(* Logix 5000 project; controller PRU vendor 1 type 14 code 107 rev 20.13; software revision 20.01; part 6 of 17 *)
(* tags used below, declared in another part *)
   AFI : BOOL;
   AlarmMaster : DINT;
   AlarmMasterDisable : BOOL;
   AlarmMasterResetTON : TIMER;
   AlarmResetPB : BOOL;
   ALL_SHUTDOWN_FAULTS_IOK : BOOL;
   DRYER : DUAL_SCREW;
   DRYER_CENTER_STARTUP_MODE : BOOL;
   DRYER_MODE_AUTO : BOOL;
   ENCODER_ERROR : REAL;
   ESR_CONTACT_1_ION : BOOL;
   ESR_CONTACT_2_ION : BOOL;
   ESTOP_PB_IOF : BOOL;   // E-STOP PUSHBUTTON IS PUSHED.
   FAULT : DINT[100];
   FAULT_TIMER : TIMER[10000];
   FS0101_ION : BOOL;   // LOW FLOW SWITCH - INLET AND DISCHARGE PURGE
   FS0102H_ION : BOOL;   // HIGH FLOW SWITCH - DISCHARGE END SHAFT SEAL
   FS0102L_ION : BOOL;   // LOW FLOW SWITCH - DISCHARGE END SHAFT SEAL
   FS0103H_ION : BOOL;   // HIGH FLOW SWITCH - CHAMBER END INLET SEALS
   FS0103L_ION : BOOL;   // LOW FLOW SWITCH - CHAMBER END INLET SEALS
   FS0201_ION : BOOL;   // LOW FLOW SWITCH - KG021 PURGE
   FS0202_ION : BOOL;   // LOW FLOW SWITCH - KG022 PURGE
   FS0203H_ION : BOOL;   // HIGH FLOW SWITCH - COOLING SHAFT SEALS
   FS0203L_ION : BOOL;   // LOW FLOW SWITCH - COOLING SHAFT SEALS
   FS0204_ION : BOOL;   // LOW FLOW SWITCH - COOLING SCREW COOLING WATER
   HMI_ALARM_RESET : BOOL;
   HMI_FINAL_SCREW_POSITION_ERROR : REAL;
   K0621_IS_LOCAL : BOOL;
   K0621_IS_REMOTE : BOOL;
   K0622_IS_LOCAL : BOOL;
   K0622_IS_REMOTE : BOOL;
   MAX_ENCODER_ERROR_MINUS_WARN : REAL;
   MAX_ENCODER_ERROR_PLUS_WARN : REAL;
   PS0101_ION : BOOL;   // PRESSURE SWITCH - CONTROL PANEL Y/Z N2 PURGE
   PS0102_ION : BOOL;   // PRESSURE SWITCH - MAIN N2 SUPPLY
   SCREWS_ENABLE_GON : BOOL;   // Dryer screw faults are ok.
   SV0101 : BOOL;
   SV0102 : BOOL;
   SV0201 : BOOL;
   SV0202 : BOOL;
   SV0203 : BOOL;
   TE0101 : REAL;
   TE0102 : REAL;
   TE0103 : REAL;
   TE0104 : REAL;
   TE0105 : REAL;
   TE0106 : REAL;
   TE0107 : REAL;
   TE0108 : REAL;
   TE0109 : REAL;
   TE0110 : REAL;
   TE0111 : REAL;
   TE0112 : REAL;
   TE0113 : REAL;
   TE0114 : REAL;
   TE0115 : REAL;
   TE0116 : REAL;
   TE0117 : REAL;
   TE0118 : REAL;
   TE0119 : REAL;
   TE0120 : REAL;
   TE0121 : REAL;
   TE0122 : REAL;
   TE0123 : REAL;
   TE0124 : REAL;
   TE0125 : REAL;
   TE0126 : REAL;
   TE0127 : REAL;
   TE0128 : REAL;
   TE0129 : REAL;
   TE0130 : REAL;
   TE0201 : REAL;
   TE0202 : REAL;
   THRESHOLD : REAL[9000];
   VFD_1_Current_Real : REAL;
   VFD_2_Current_Real : REAL;
   VFD_3_Current_Real : REAL;
   VFDS_BON : BOOL;   // DRYER VFDs HAVE BEEN COMMANDED ON FOR 1 SECOND.
   WARNA_IOK : BOOL;
   WARND_IOK : BOOL;
   WARNE_IOK : BOOL;
   WIPE_ACTUAL : REAL;
(* MainProgram, continued *)

ROUTINE A4_Alarms_General   (* ladder *)
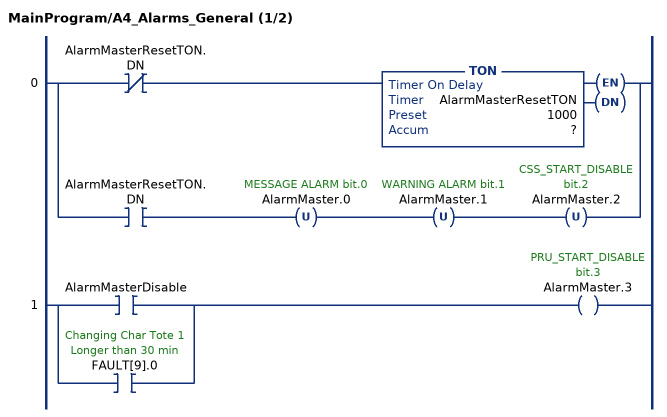
   0: [XIO(AlarmMasterResetTON.DN) TON(AlarmMasterResetTON,?,?) ,XIC(AlarmMasterResetTON.DN) OTU(AlarmMaster.0) OTU(AlarmMaster.1) OTU(AlarmMaster.2) ];
   1: [XIC(AlarmMasterDisable) ,XIC(FAULT[9].0) ]OTE(AlarmMaster.3);
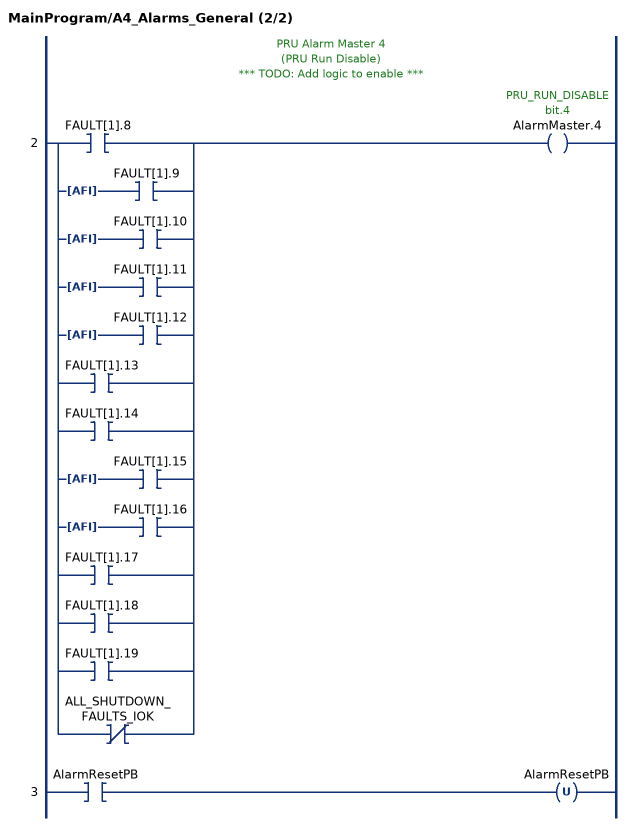
   // PRU Alarm Master 4
   // (PRU Run Disable)
   // *** TODO: Add logic to enable ***
   2: [XIC(FAULT[1].8) ,AFI() XIC(FAULT[1].9) ,AFI() XIC(FAULT[1].10) ,AFI() XIC(FAULT[1].11) ,AFI() XIC(FAULT[1].12) ,XIC(FAULT[1].13) ,XIC(FAULT[1].14) ,AFI() XIC(FAULT[1].15) ,AFI() XIC(FAULT[1].16) ,XIC(FAULT[1].17) ,XIC(FAULT[1].18) ,XIC(FAULT[1].19) ,XIO(ALL_SHUTDOWN_FAULTS_IOK) ]OTE(AlarmMaster.4);
   3: XIC(AlarmResetPB)OTU(AlarmResetPB);
END_ROUTINE

ROUTINE B00_WARN_A_100   (* ladder *)
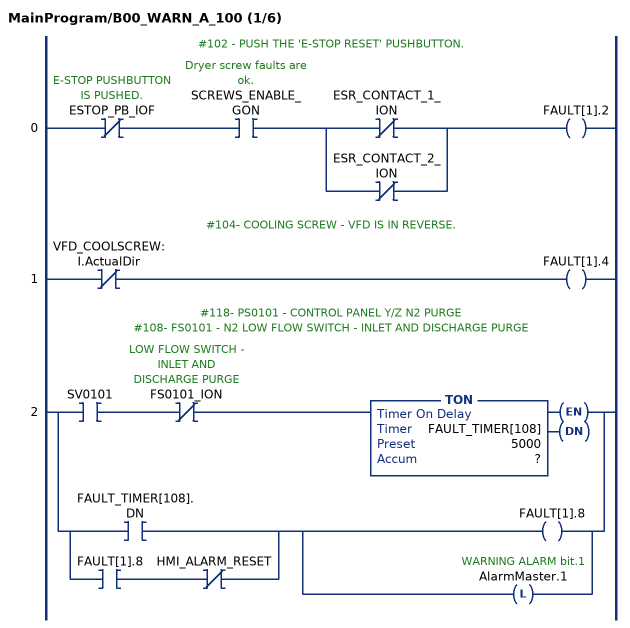
   // #102 - PUSH THE 'E-STOP RESET' PUSHBUTTON.
   0: XIO(ESTOP_PB_IOF)XIC(SCREWS_ENABLE_GON)[XIO(ESR_CONTACT_1_ION) ,XIO(ESR_CONTACT_2_ION) ]OTE(FAULT[1].2);
   // #104- COOLING SCREW - VFD IS IN REVERSE.
   1: XIO(VFD_COOLSCREW:I.ActualDir)OTE(FAULT[1].4);
   // #118- PS0101 - CONTROL PANEL Y/Z N2 PURGE
   // #108- FS0101 - N2 LOW FLOW SWITCH - INLET AND DISCHARGE PURGE
   2: [XIC(SV0101) XIO(FS0101_ION) TON(FAULT_TIMER[108],?,?) ,[XIC(FAULT_TIMER[108].DN) ,XIC(FAULT[1].8) XIO(HMI_ALARM_RESET) ] [OTE(FAULT[1].8) ,OTL(AlarmMaster.1) ] ];
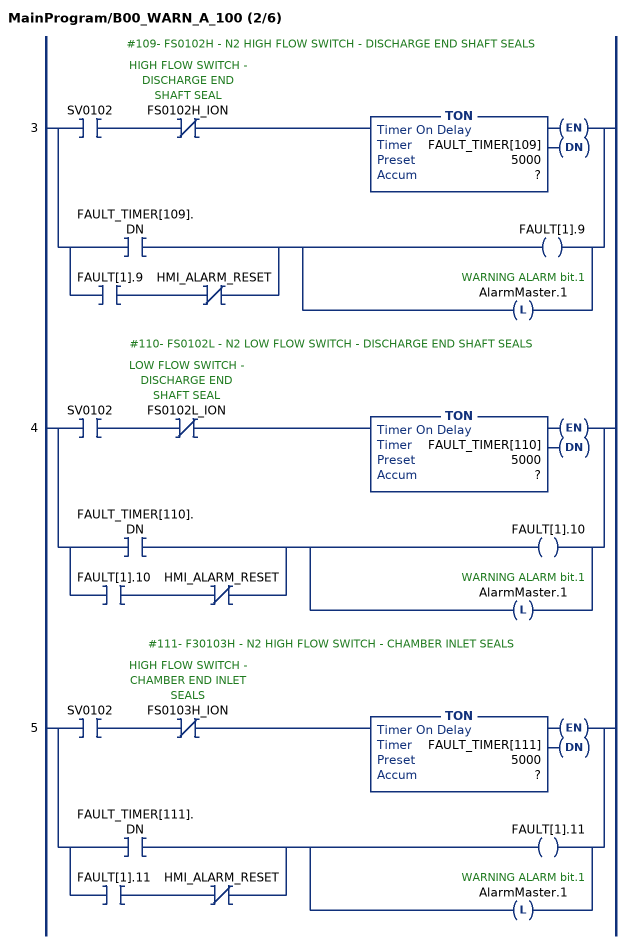
   // #109- FS0102H - N2 HIGH FLOW SWITCH - DISCHARGE END SHAFT SEALS
   3: [XIC(SV0102) XIO(FS0102H_ION) TON(FAULT_TIMER[109],?,?) ,[XIC(FAULT_TIMER[109].DN) ,XIC(FAULT[1].9) XIO(HMI_ALARM_RESET) ] [OTE(FAULT[1].9) ,OTL(AlarmMaster.1) ] ];
   // #110- FS0102L - N2 LOW FLOW SWITCH - DISCHARGE END SHAFT SEALS
   4: [XIC(SV0102) XIO(FS0102L_ION) TON(FAULT_TIMER[110],?,?) ,[XIC(FAULT_TIMER[110].DN) ,XIC(FAULT[1].10) XIO(HMI_ALARM_RESET) ] [OTE(FAULT[1].10) ,OTL(AlarmMaster.1) ] ];
   // #111- F30103H - N2 HIGH FLOW SWITCH - CHAMBER INLET SEALS
   5: [XIC(SV0102) XIO(FS0103H_ION) TON(FAULT_TIMER[111],?,?) ,[XIC(FAULT_TIMER[111].DN) ,XIC(FAULT[1].11) XIO(HMI_ALARM_RESET) ] [OTE(FAULT[1].11) ,OTL(AlarmMaster.1) ] ];
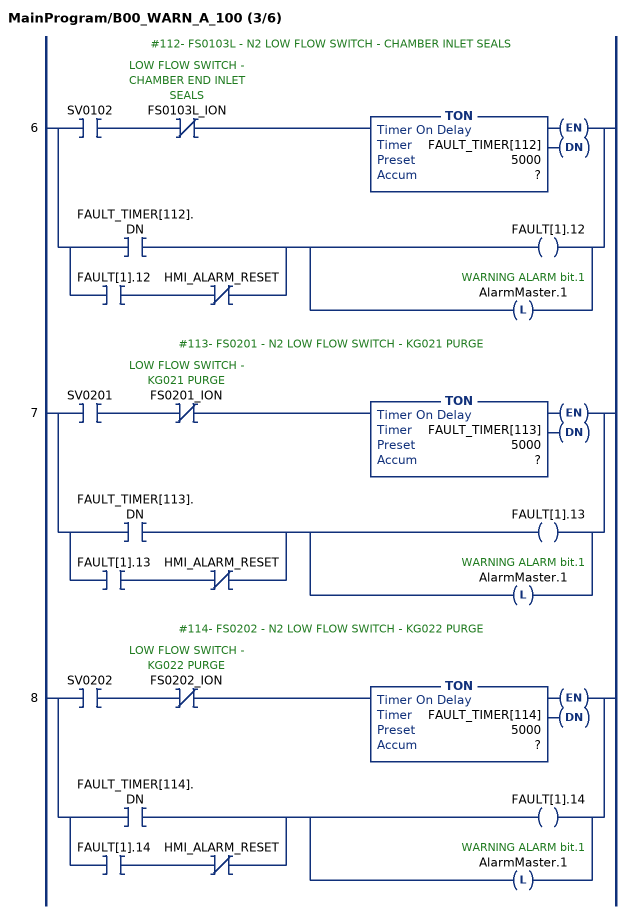
   // #112- FS0103L - N2 LOW FLOW SWITCH - CHAMBER INLET SEALS
   6: [XIC(SV0102) XIO(FS0103L_ION) TON(FAULT_TIMER[112],?,?) ,[XIC(FAULT_TIMER[112].DN) ,XIC(FAULT[1].12) XIO(HMI_ALARM_RESET) ] [OTE(FAULT[1].12) ,OTL(AlarmMaster.1) ] ];
   // #113- FS0201 - N2 LOW FLOW SWITCH - KG021 PURGE
   7: [XIC(SV0201) XIO(FS0201_ION) TON(FAULT_TIMER[113],?,?) ,[XIC(FAULT_TIMER[113].DN) ,XIC(FAULT[1].13) XIO(HMI_ALARM_RESET) ] [OTE(FAULT[1].13) ,OTL(AlarmMaster.1) ] ];
   // #114- FS0202 - N2 LOW FLOW SWITCH - KG022 PURGE
   8: [XIC(SV0202) XIO(FS0202_ION) TON(FAULT_TIMER[114],?,?) ,[XIC(FAULT_TIMER[114].DN) ,XIC(FAULT[1].14) XIO(HMI_ALARM_RESET) ] [OTE(FAULT[1].14) ,OTL(AlarmMaster.1) ] ];
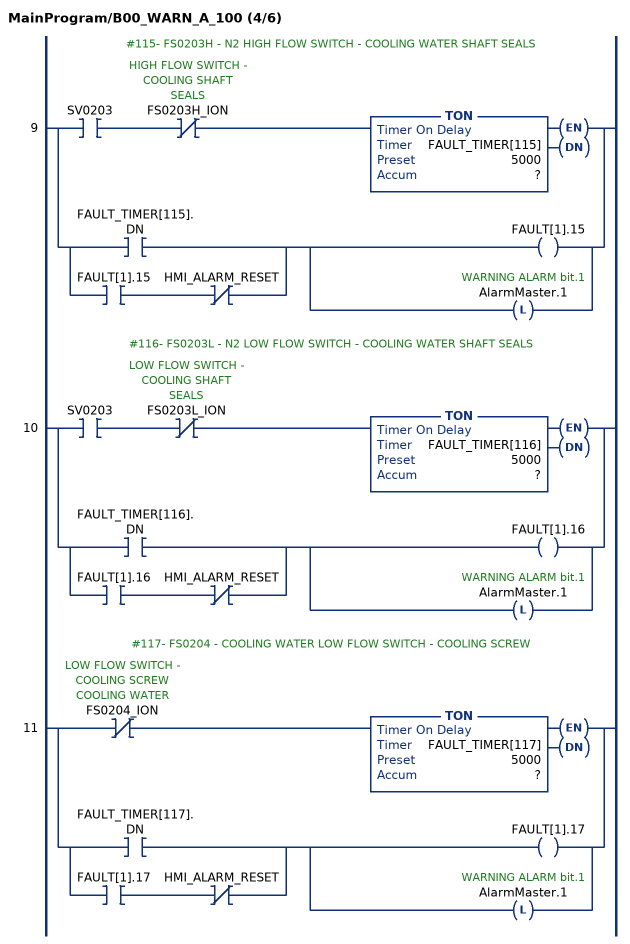
   // #115- FS0203H - N2 HIGH FLOW SWITCH - COOLING WATER SHAFT SEALS
   9: [XIC(SV0203) XIO(FS0203H_ION) TON(FAULT_TIMER[115],?,?) ,[XIC(FAULT_TIMER[115].DN) ,XIC(FAULT[1].15) XIO(HMI_ALARM_RESET) ] [OTE(FAULT[1].15) ,OTL(AlarmMaster.1) ] ];
   // #116- FS0203L - N2 LOW FLOW SWITCH - COOLING WATER SHAFT SEALS
   10: [XIC(SV0203) XIO(FS0203L_ION) TON(FAULT_TIMER[116],?,?) ,[XIC(FAULT_TIMER[116].DN) ,XIC(FAULT[1].16) XIO(HMI_ALARM_RESET) ] [OTE(FAULT[1].16) ,OTL(AlarmMaster.1) ] ];
   // #117- FS0204 - COOLING WATER LOW FLOW SWITCH - COOLING SCREW
   11: [XIO(FS0204_ION) TON(FAULT_TIMER[117],?,?) ,[XIC(FAULT_TIMER[117].DN) ,XIC(FAULT[1].17) XIO(HMI_ALARM_RESET) ] [OTE(FAULT[1].17) ,OTL(AlarmMaster.1) ] ];
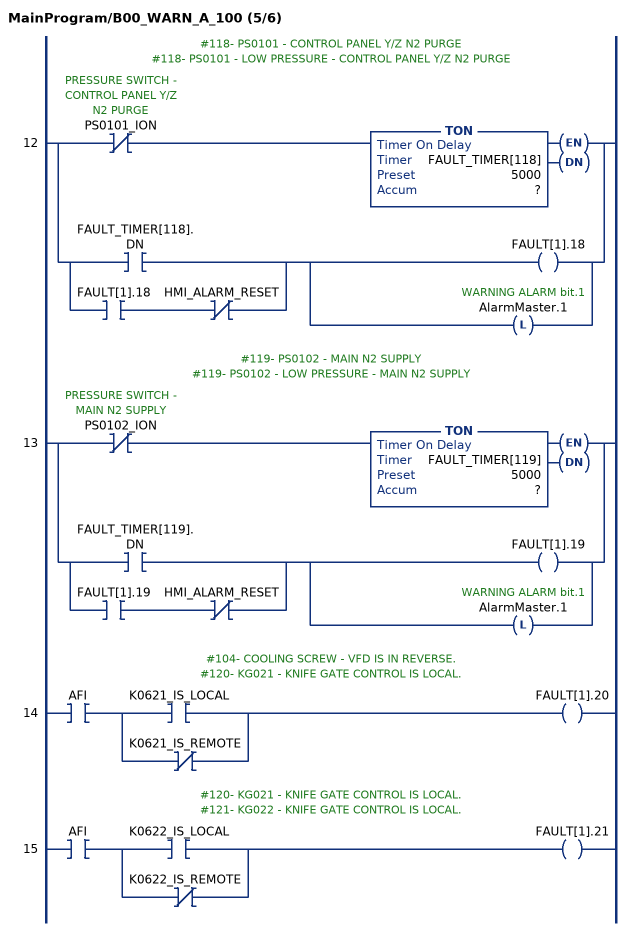
   // #118- PS0101 - CONTROL PANEL Y/Z N2 PURGE
   // #118- PS0101 - LOW PRESSURE - CONTROL PANEL Y/Z N2 PURGE
   12: [XIO(PS0101_ION) TON(FAULT_TIMER[118],?,?) ,[XIC(FAULT_TIMER[118].DN) ,XIC(FAULT[1].18) XIO(HMI_ALARM_RESET) ] [OTE(FAULT[1].18) ,OTL(AlarmMaster.1) ] ];
   // #119- PS0102 - MAIN N2 SUPPLY
   // #119- PS0102 - LOW PRESSURE - MAIN N2 SUPPLY
   13: [XIO(PS0102_ION) TON(FAULT_TIMER[119],?,?) ,[XIC(FAULT_TIMER[119].DN) ,XIC(FAULT[1].19) XIO(HMI_ALARM_RESET) ] [OTE(FAULT[1].19) ,OTL(AlarmMaster.1) ] ];
   // #104- COOLING SCREW - VFD IS IN REVERSE.
   // #120- KG021 - KNIFE GATE CONTROL IS LOCAL.
   14: XIC(AFI)[XIC(K0621_IS_LOCAL) ,XIO(K0621_IS_REMOTE) ]OTE(FAULT[1].20);
   // #120- KG021 - KNIFE GATE CONTROL IS LOCAL.
   // #121- KG022 - KNIFE GATE CONTROL IS LOCAL.
   15: XIC(AFI)[XIC(K0622_IS_LOCAL) ,XIO(K0622_IS_REMOTE) ]OTE(FAULT[1].21);
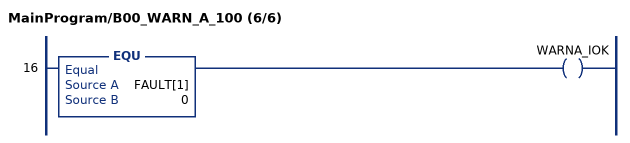
   16: EQU(FAULT[1],0)OTE(WARNA_IOK);
END_ROUTINE

ROUTINE B00_WARN_D_400_CURRENT   (* ladder *)
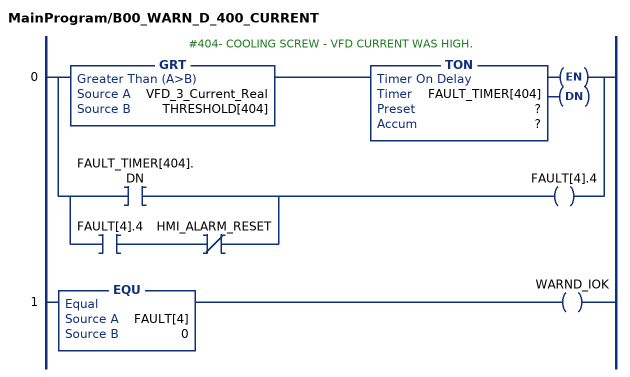
   // #404- COOLING SCREW - VFD CURRENT WAS HIGH.
   0: [GRT(VFD_3_Current_Real,THRESHOLD[404]) TON(FAULT_TIMER[404],?,?) ,[XIC(FAULT_TIMER[404].DN) ,XIC(FAULT[4].4) XIO(HMI_ALARM_RESET) ] OTE(FAULT[4].4) ];
   1: EQU(FAULT[4],0)OTE(WARND_IOK);
END_ROUTINE

ROUTINE B00_WARN_E_500_DRYER   (* ladder *)
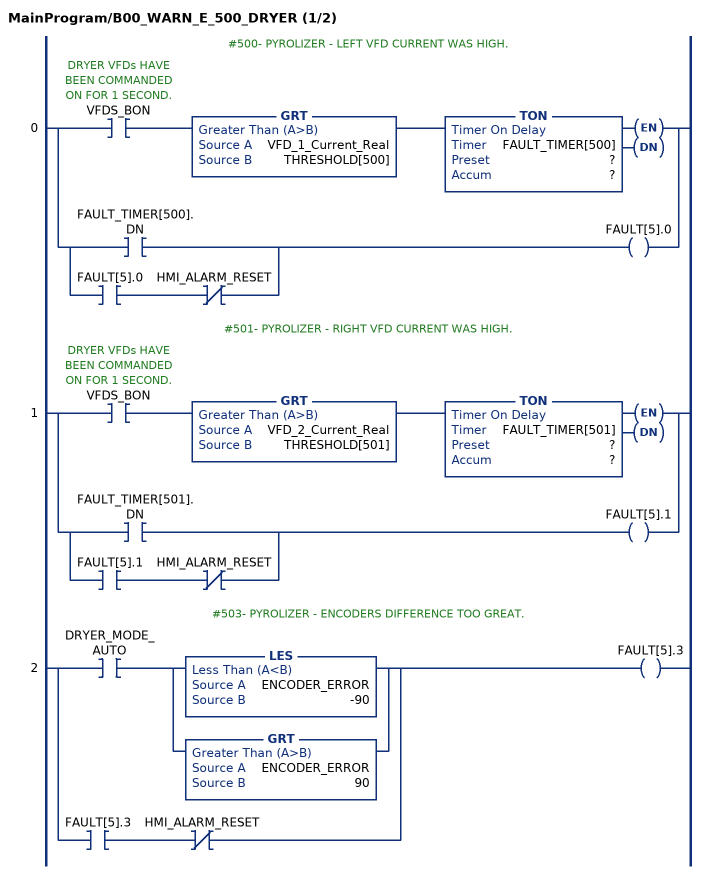
   // #500- PYROLIZER - LEFT VFD CURRENT WAS HIGH.
   0: [XIC(VFDS_BON) GRT(VFD_1_Current_Real,THRESHOLD[500]) TON(FAULT_TIMER[500],?,?) ,[XIC(FAULT_TIMER[500].DN) ,XIC(FAULT[5].0) XIO(HMI_ALARM_RESET) ] OTE(FAULT[5].0) ];
   // #501- PYROLIZER - RIGHT VFD CURRENT WAS HIGH.
   1: [XIC(VFDS_BON) GRT(VFD_2_Current_Real,THRESHOLD[501]) TON(FAULT_TIMER[501],?,?) ,[XIC(FAULT_TIMER[501].DN) ,XIC(FAULT[5].1) XIO(HMI_ALARM_RESET) ] OTE(FAULT[5].1) ];
   // #503- PYROLIZER - ENCODERS DIFFERENCE TOO GREAT.
   2: [XIC(DRYER_MODE_AUTO) [LES(ENCODER_ERROR,-90) ,GRT(ENCODER_ERROR,90) ] ,XIC(FAULT[5].3) XIO(HMI_ALARM_RESET) ]OTE(FAULT[5].3);
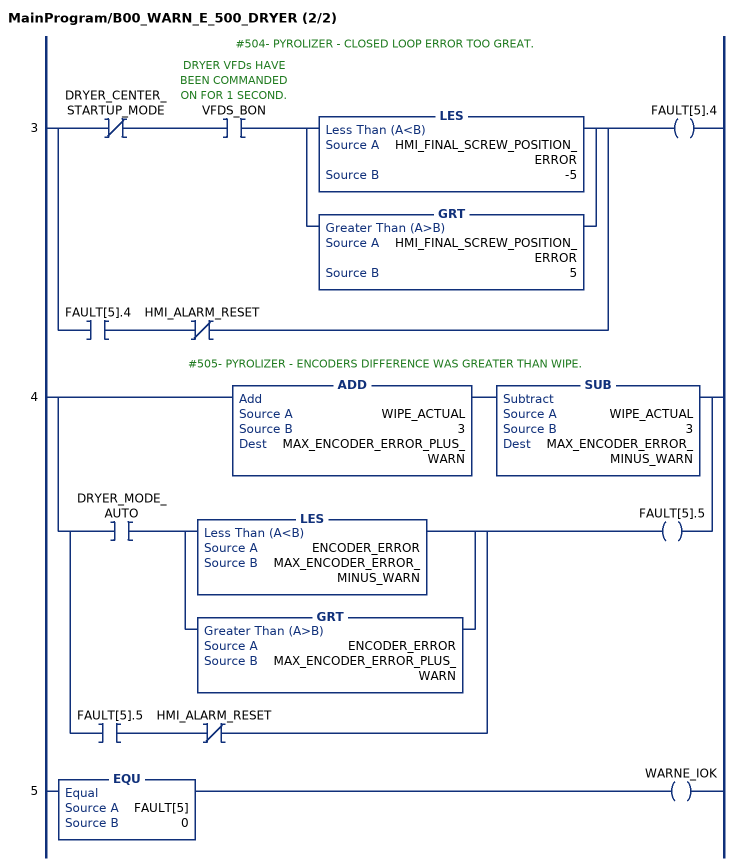
   // #504- PYROLIZER - CLOSED LOOP ERROR TOO GREAT.
   3: [XIO(DRYER_CENTER_STARTUP_MODE) XIC(VFDS_BON) [LES(HMI_FINAL_SCREW_POSITION_ERROR,-5) ,GRT(HMI_FINAL_SCREW_POSITION_ERROR,5) ] ,XIC(FAULT[5].4) XIO(HMI_ALARM_RESET) ]OTE(FAULT[5].4);
   // #505- PYROLIZER - ENCODERS DIFFERENCE WAS GREATER THAN WIPE.
   4: [ADD(WIPE_ACTUAL,3,MAX_ENCODER_ERROR_PLUS_WARN) SUB(WIPE_ACTUAL,3,MAX_ENCODER_ERROR_MINUS_WARN) ,[XIC(DRYER_MODE_AUTO) [LES(ENCODER_ERROR,MAX_ENCODER_ERROR_MINUS_WARN) ,GRT(ENCODER_ERROR,MAX_ENCODER_ERROR_PLUS_WARN) ] ,XIC(FAULT[5].5) XIO(HMI_ALARM_RESET) ] OTE(FAULT[5].5) ];
   5: EQU(FAULT[5],0)OTE(WARNE_IOK);
END_ROUTINE

ROUTINE B00_WARN_F_600_HI_TEMP   (* ladder *)
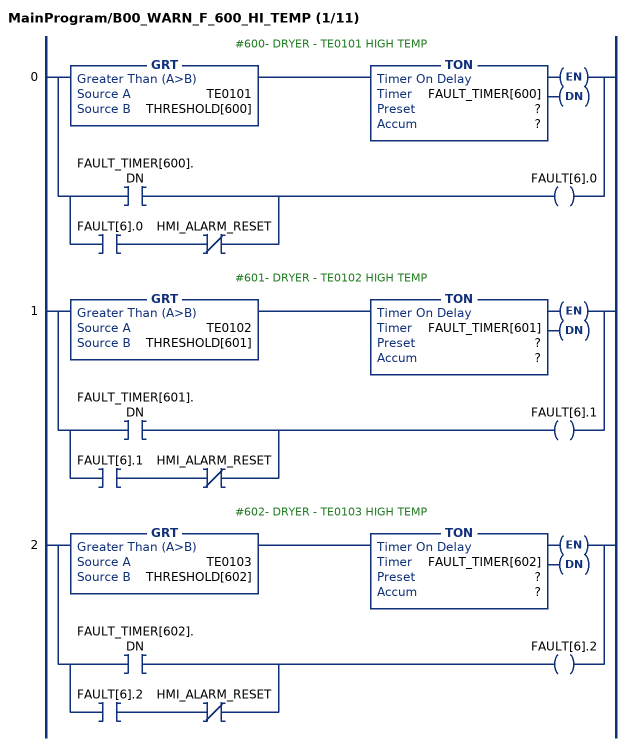
   // #600- DRYER - TE0101 HIGH TEMP
   0: [GRT(TE0101,THRESHOLD[600]) TON(FAULT_TIMER[600],?,?) ,[XIC(FAULT_TIMER[600].DN) ,XIC(FAULT[6].0) XIO(HMI_ALARM_RESET) ] OTE(FAULT[6].0) ];
   // #601- DRYER - TE0102 HIGH TEMP
   1: [GRT(TE0102,THRESHOLD[601]) TON(FAULT_TIMER[601],?,?) ,[XIC(FAULT_TIMER[601].DN) ,XIC(FAULT[6].1) XIO(HMI_ALARM_RESET) ] OTE(FAULT[6].1) ];
   // #602- DRYER - TE0103 HIGH TEMP
   2: [GRT(TE0103,THRESHOLD[602]) TON(FAULT_TIMER[602],?,?) ,[XIC(FAULT_TIMER[602].DN) ,XIC(FAULT[6].2) XIO(HMI_ALARM_RESET) ] OTE(FAULT[6].2) ];
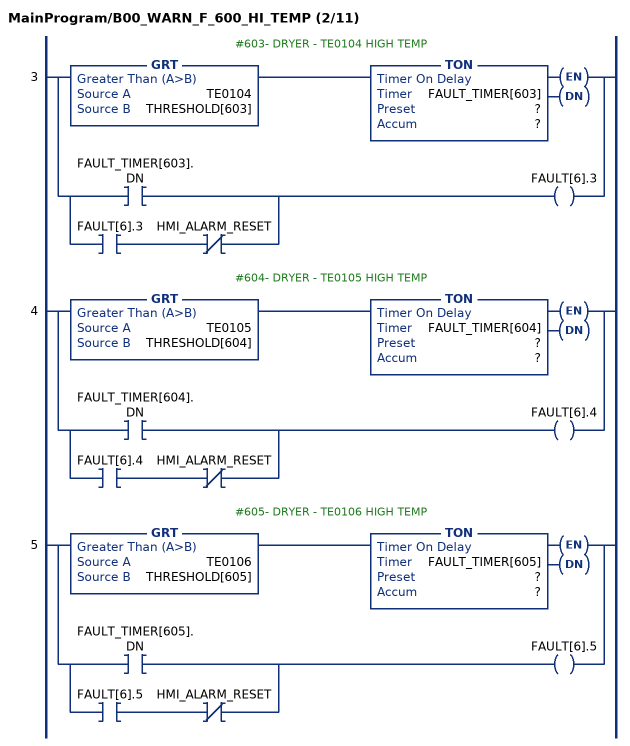
   // #603- DRYER - TE0104 HIGH TEMP
   3: [GRT(TE0104,THRESHOLD[603]) TON(FAULT_TIMER[603],?,?) ,[XIC(FAULT_TIMER[603].DN) ,XIC(FAULT[6].3) XIO(HMI_ALARM_RESET) ] OTE(FAULT[6].3) ];
   // #604- DRYER - TE0105 HIGH TEMP
   4: [GRT(TE0105,THRESHOLD[604]) TON(FAULT_TIMER[604],?,?) ,[XIC(FAULT_TIMER[604].DN) ,XIC(FAULT[6].4) XIO(HMI_ALARM_RESET) ] OTE(FAULT[6].4) ];
   // #605- DRYER - TE0106 HIGH TEMP
   5: [GRT(TE0106,THRESHOLD[605]) TON(FAULT_TIMER[605],?,?) ,[XIC(FAULT_TIMER[605].DN) ,XIC(FAULT[6].5) XIO(HMI_ALARM_RESET) ] OTE(FAULT[6].5) ];
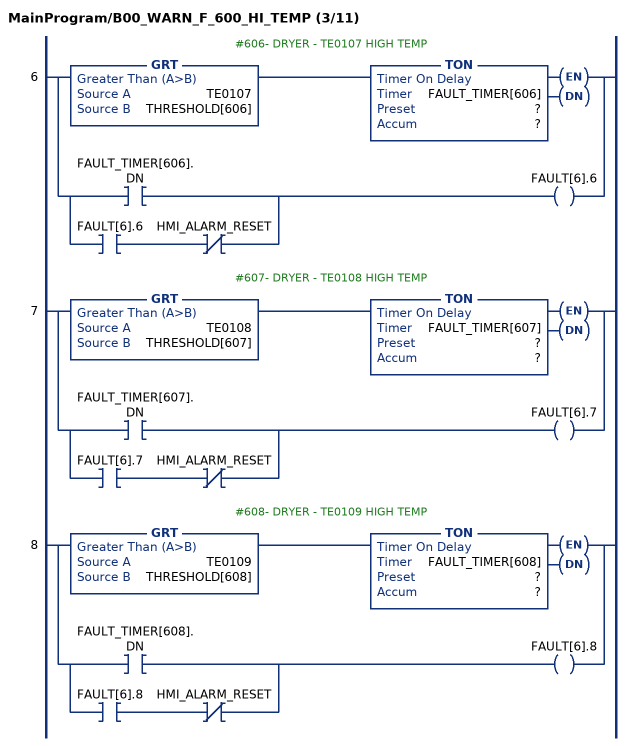
   // #606- DRYER - TE0107 HIGH TEMP
   6: [GRT(TE0107,THRESHOLD[606]) TON(FAULT_TIMER[606],?,?) ,[XIC(FAULT_TIMER[606].DN) ,XIC(FAULT[6].6) XIO(HMI_ALARM_RESET) ] OTE(FAULT[6].6) ];
   // #607- DRYER - TE0108 HIGH TEMP
   7: [GRT(TE0108,THRESHOLD[607]) TON(FAULT_TIMER[607],?,?) ,[XIC(FAULT_TIMER[607].DN) ,XIC(FAULT[6].7) XIO(HMI_ALARM_RESET) ] OTE(FAULT[6].7) ];
   // #608- DRYER - TE0109 HIGH TEMP
   8: [GRT(TE0109,THRESHOLD[608]) TON(FAULT_TIMER[608],?,?) ,[XIC(FAULT_TIMER[608].DN) ,XIC(FAULT[6].8) XIO(HMI_ALARM_RESET) ] OTE(FAULT[6].8) ];
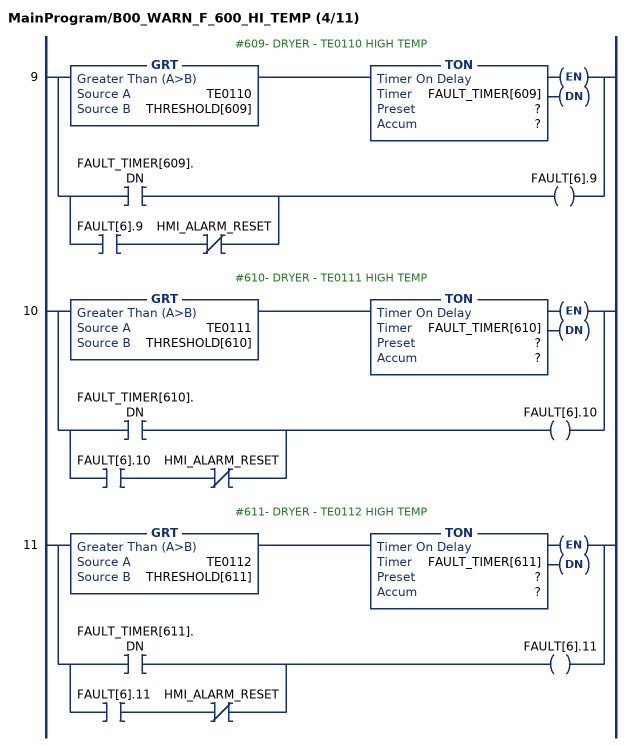
   // #609- DRYER - TE0110 HIGH TEMP
   9: [GRT(TE0110,THRESHOLD[609]) TON(FAULT_TIMER[609],?,?) ,[XIC(FAULT_TIMER[609].DN) ,XIC(FAULT[6].9) XIO(HMI_ALARM_RESET) ] OTE(FAULT[6].9) ];
   // #610- DRYER - TE0111 HIGH TEMP
   10: [GRT(TE0111,THRESHOLD[610]) TON(FAULT_TIMER[610],?,?) ,[XIC(FAULT_TIMER[610].DN) ,XIC(FAULT[6].10) XIO(HMI_ALARM_RESET) ] OTE(FAULT[6].10) ];
   // #611- DRYER - TE0112 HIGH TEMP
   11: [GRT(TE0112,THRESHOLD[611]) TON(FAULT_TIMER[611],?,?) ,[XIC(FAULT_TIMER[611].DN) ,XIC(FAULT[6].11) XIO(HMI_ALARM_RESET) ] OTE(FAULT[6].11) ];
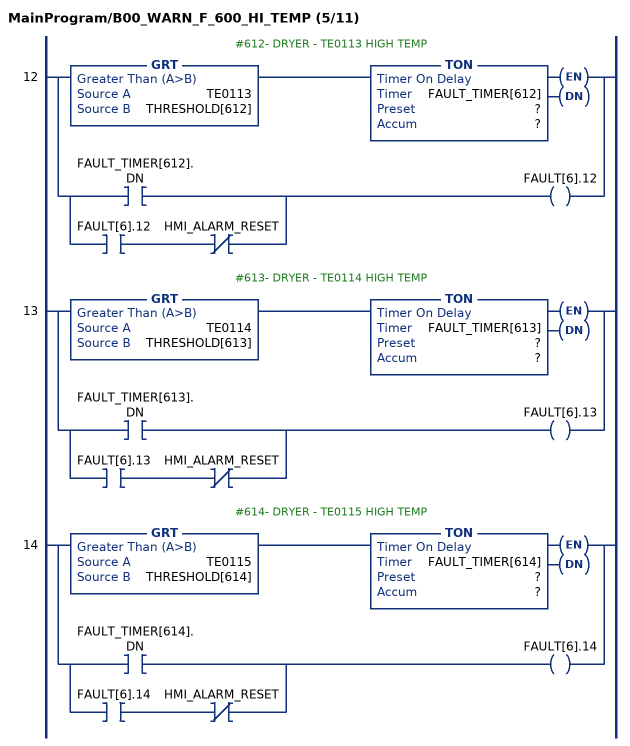
   // #612- DRYER - TE0113 HIGH TEMP
   12: [GRT(TE0113,THRESHOLD[612]) TON(FAULT_TIMER[612],?,?) ,[XIC(FAULT_TIMER[612].DN) ,XIC(FAULT[6].12) XIO(HMI_ALARM_RESET) ] OTE(FAULT[6].12) ];
   // #613- DRYER - TE0114 HIGH TEMP
   13: [GRT(TE0114,THRESHOLD[613]) TON(FAULT_TIMER[613],?,?) ,[XIC(FAULT_TIMER[613].DN) ,XIC(FAULT[6].13) XIO(HMI_ALARM_RESET) ] OTE(FAULT[6].13) ];
   // #614- DRYER - TE0115 HIGH TEMP
   14: [GRT(TE0115,THRESHOLD[614]) TON(FAULT_TIMER[614],?,?) ,[XIC(FAULT_TIMER[614].DN) ,XIC(FAULT[6].14) XIO(HMI_ALARM_RESET) ] OTE(FAULT[6].14) ];
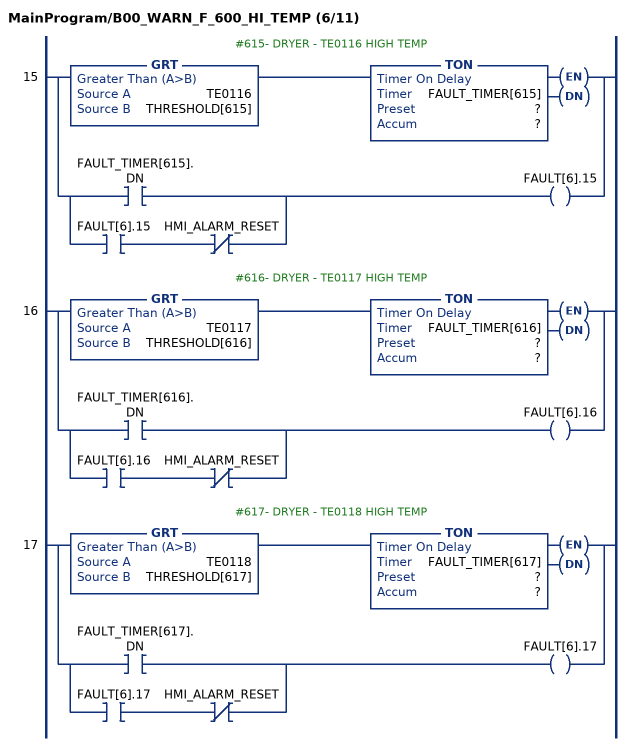
   // #615- DRYER - TE0116 HIGH TEMP
   15: [GRT(TE0116,THRESHOLD[615]) TON(FAULT_TIMER[615],?,?) ,[XIC(FAULT_TIMER[615].DN) ,XIC(FAULT[6].15) XIO(HMI_ALARM_RESET) ] OTE(FAULT[6].15) ];
   // #616- DRYER - TE0117 HIGH TEMP
   16: [GRT(TE0117,THRESHOLD[616]) TON(FAULT_TIMER[616],?,?) ,[XIC(FAULT_TIMER[616].DN) ,XIC(FAULT[6].16) XIO(HMI_ALARM_RESET) ] OTE(FAULT[6].16) ];
   // #617- DRYER - TE0118 HIGH TEMP
   17: [GRT(TE0118,THRESHOLD[617]) TON(FAULT_TIMER[617],?,?) ,[XIC(FAULT_TIMER[617].DN) ,XIC(FAULT[6].17) XIO(HMI_ALARM_RESET) ] OTE(FAULT[6].17) ];
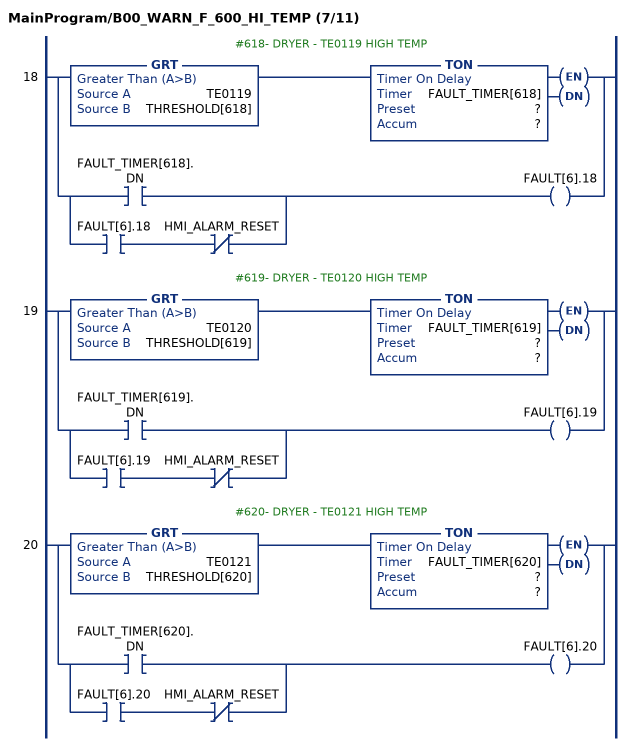
   // #618- DRYER - TE0119 HIGH TEMP
   18: [GRT(TE0119,THRESHOLD[618]) TON(FAULT_TIMER[618],?,?) ,[XIC(FAULT_TIMER[618].DN) ,XIC(FAULT[6].18) XIO(HMI_ALARM_RESET) ] OTE(FAULT[6].18) ];
   // #619- DRYER - TE0120 HIGH TEMP
   19: [GRT(TE0120,THRESHOLD[619]) TON(FAULT_TIMER[619],?,?) ,[XIC(FAULT_TIMER[619].DN) ,XIC(FAULT[6].19) XIO(HMI_ALARM_RESET) ] OTE(FAULT[6].19) ];
   // #620- DRYER - TE0121 HIGH TEMP
   20: [GRT(TE0121,THRESHOLD[620]) TON(FAULT_TIMER[620],?,?) ,[XIC(FAULT_TIMER[620].DN) ,XIC(FAULT[6].20) XIO(HMI_ALARM_RESET) ] OTE(FAULT[6].20) ];
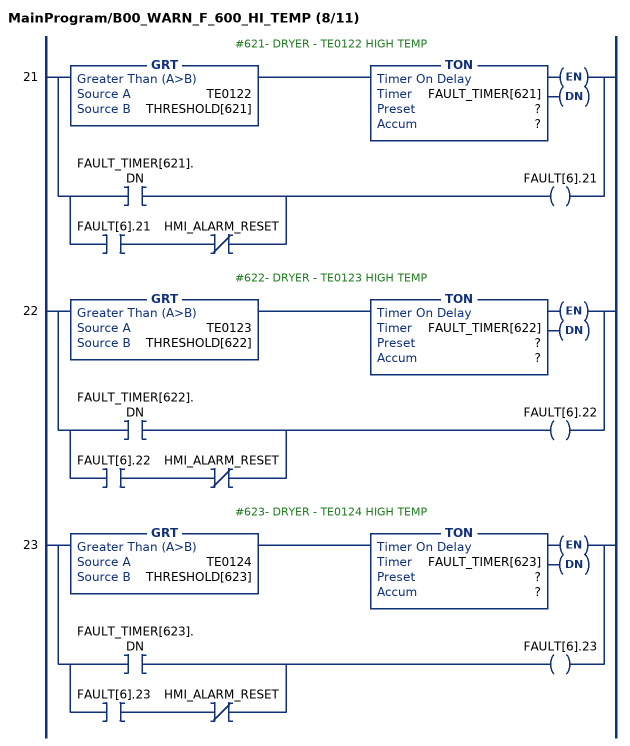
   // #621- DRYER - TE0122 HIGH TEMP
   21: [GRT(TE0122,THRESHOLD[621]) TON(FAULT_TIMER[621],?,?) ,[XIC(FAULT_TIMER[621].DN) ,XIC(FAULT[6].21) XIO(HMI_ALARM_RESET) ] OTE(FAULT[6].21) ];
   // #622- DRYER - TE0123 HIGH TEMP
   22: [GRT(TE0123,THRESHOLD[622]) TON(FAULT_TIMER[622],?,?) ,[XIC(FAULT_TIMER[622].DN) ,XIC(FAULT[6].22) XIO(HMI_ALARM_RESET) ] OTE(FAULT[6].22) ];
   // #623- DRYER - TE0124 HIGH TEMP
   23: [GRT(TE0124,THRESHOLD[623]) TON(FAULT_TIMER[623],?,?) ,[XIC(FAULT_TIMER[623].DN) ,XIC(FAULT[6].23) XIO(HMI_ALARM_RESET) ] OTE(FAULT[6].23) ];
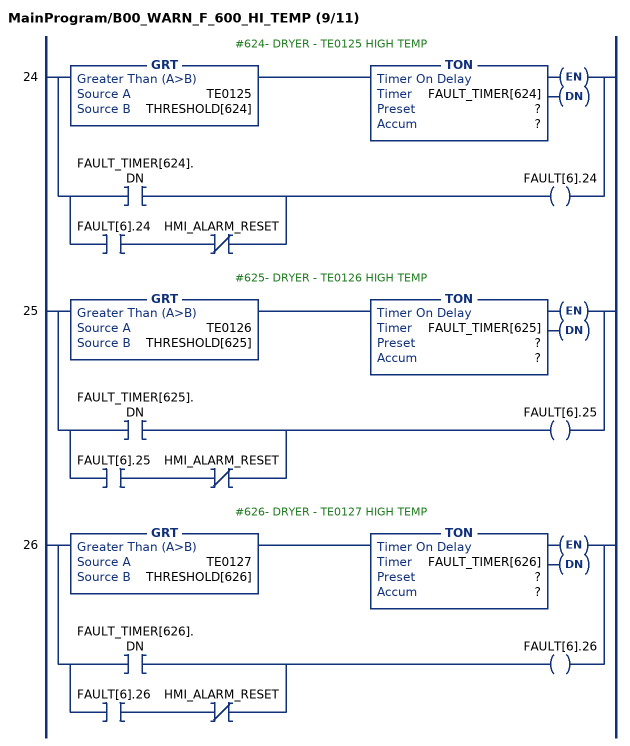
   // #624- DRYER - TE0125 HIGH TEMP
   24: [GRT(TE0125,THRESHOLD[624]) TON(FAULT_TIMER[624],?,?) ,[XIC(FAULT_TIMER[624].DN) ,XIC(FAULT[6].24) XIO(HMI_ALARM_RESET) ] OTE(FAULT[6].24) ];
   // #625- DRYER - TE0126 HIGH TEMP
   25: [GRT(TE0126,THRESHOLD[625]) TON(FAULT_TIMER[625],?,?) ,[XIC(FAULT_TIMER[625].DN) ,XIC(FAULT[6].25) XIO(HMI_ALARM_RESET) ] OTE(FAULT[6].25) ];
   // #626- DRYER - TE0127 HIGH TEMP
   26: [GRT(TE0127,THRESHOLD[626]) TON(FAULT_TIMER[626],?,?) ,[XIC(FAULT_TIMER[626].DN) ,XIC(FAULT[6].26) XIO(HMI_ALARM_RESET) ] OTE(FAULT[6].26) ];
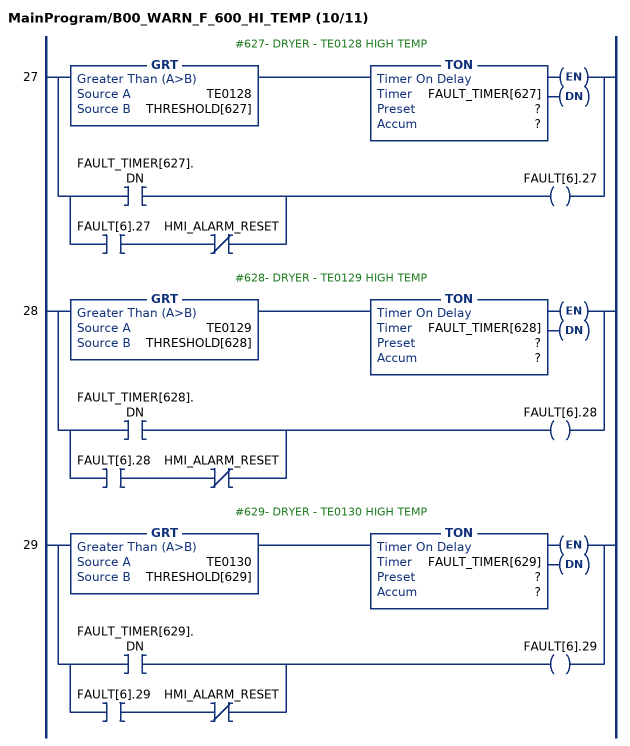
   // #627- DRYER - TE0128 HIGH TEMP
   27: [GRT(TE0128,THRESHOLD[627]) TON(FAULT_TIMER[627],?,?) ,[XIC(FAULT_TIMER[627].DN) ,XIC(FAULT[6].27) XIO(HMI_ALARM_RESET) ] OTE(FAULT[6].27) ];
   // #628- DRYER - TE0129 HIGH TEMP
   28: [GRT(TE0129,THRESHOLD[628]) TON(FAULT_TIMER[628],?,?) ,[XIC(FAULT_TIMER[628].DN) ,XIC(FAULT[6].28) XIO(HMI_ALARM_RESET) ] OTE(FAULT[6].28) ];
   // #629- DRYER - TE0130 HIGH TEMP
   29: [GRT(TE0130,THRESHOLD[629]) TON(FAULT_TIMER[629],?,?) ,[XIC(FAULT_TIMER[629].DN) ,XIC(FAULT[6].29) XIO(HMI_ALARM_RESET) ] OTE(FAULT[6].29) ];
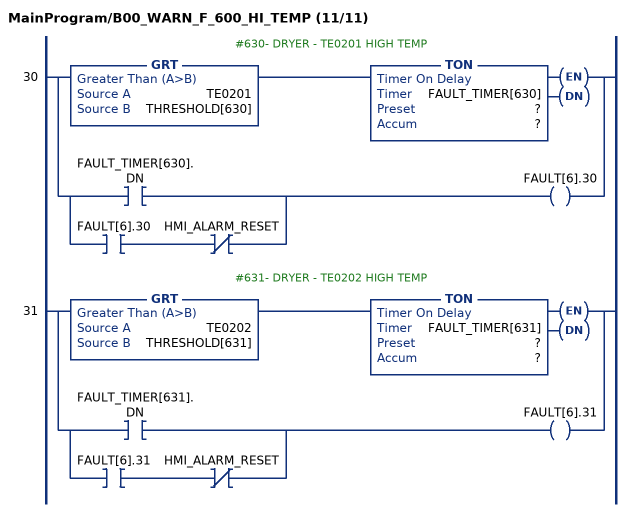
   // #630- DRYER - TE0201 HIGH TEMP
   30: [GRT(TE0201,THRESHOLD[630]) TON(FAULT_TIMER[630],?,?) ,[XIC(FAULT_TIMER[630].DN) ,XIC(FAULT[6].30) XIO(HMI_ALARM_RESET) ] OTE(FAULT[6].30) ];
   // #631- DRYER - TE0202 HIGH TEMP
   31: [GRT(TE0202,THRESHOLD[631]) TON(FAULT_TIMER[631],?,?) ,[XIC(FAULT_TIMER[631].DN) ,XIC(FAULT[6].31) XIO(HMI_ALARM_RESET) ] OTE(FAULT[6].31) ];
END_ROUTINE
